(*
SPDX-FileCopyrightText: © 2026 Oleksandr Tiutyk <trofimich@gmail.com>
SPDX-License-Identifier: MIT
License: https://opensource.org/license/mit
*)

//!<param name="CountObjectStatistics">Indicates if object creating and deleting counted in ObjectStatistics</param>

{attribute 'qualified_only'}
VAR_GLOBAL PERSISTENT
	{attribute 'OPC.UA.DA' := '1'}	
	
	CountObjectStatistics : BOOL;
END_VAR

(* stored: Version 1.1.0.1
   GVL ObjectStatisticsSettings: Id {7f924c5f-0383-4dfc-a181-e3d9714446b9} *)
